Omron CX-Programmer project NewProject (CX-Programmer 9.73)

# PLC NewPLC1: CP1E N20

## Global symbols (name address type ; comment)
0.01 BOOL  ; PB STOP
0.11 BOOL  ; PB START
100.00 BOOL  ; OUTPUT
100.01 BOOL  ; OUTPUT
100.02 BOOL  ; OUTPUT
100.07 BOOL  ; OUTPUT
200.01 BOOL  ; RELAY

## Program NewProgram1 (cyclic task 0)

### Section Section1

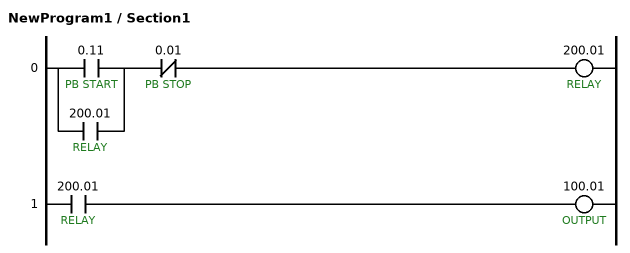
; rung 0
LD 0.11  ; PB START
OR 200.01  ; RELAY
ANDNOT 0.01  ; PB STOP
OUT 200.01  ; RELAY
; rung 1
LD 200.01  ; RELAY
OUT 100.01  ; OUTPUT

### Section END
; rung 0
END(001)